KUKA KRL program: chk_w6_grp4_opn.src

&ACCESS RV4
&COMMENT Check GRP AXOR Z4 OPEN
DEF chk_w6_grp4_opn( )

; Check gripper axor OPEN Z4.1
;//---- Start User-------

$TIMER[10] = 0
$TIMER_STOP[10] = FALSE

WAIT FOR ($IN[499])
WAIT FOR (NOT $IN[500])

$TIMER_STOP[10] = TRUE
$TIMER[10] = 0

;//---- End User---------
END
